TYPE ST_Gyroscope :
STRUCT
	Pitch: INT;
	Yaw: INT;
	Roll: INT;
END_STRUCT
END_TYPE

(* stored: Version 1.1.0.1
   DUT ST_Gyroscope: Id {18138b89-cf57-409e-a883-6a58c1af160a} *)
